FUNCTION_BLOCK FB_DetectorCapacitivo EXTENDS FB_Module
(*
ESTACIONES DE DETECCIÓN DE MATERIAL - Manual de usuario #32/28

La detección de las tapas realizadas en nylon, ha de llevarse a cabo por tanto 
a través de otro sensor. Para ello se ha dispuesto un detector capacitivo, 
que a diferencia del anterior proporciona una señal al PLC cuando se sitúa 
en su rango de detección una pieza de cualquier material 

*)
VAR_INPUT

END_VAR
VAR_OUTPUT
	CapacidadDetectada: BOOL;
	TapaMetalica: BOOL;
END_VAR
VAR
END_VAR

// Falta este módulo

END_FUNCTION_BLOCK

(* stored: Version 1.1.0.1, ProductVersion 3.1.4024.11
   POU FB_DetectorCapacitivo: Id {51b32ed3-45d8-4130-8ade-74f05fee5c33}, SpecialFunc None *)
